// TIA Portal V20 export
VAR_GLOBAL   // PLC tag table "ConvConstantD1"
END_VAR
VAR_GLOBAL CONSTANT   // user constants
   minD1 : Int := 4001;
   maxD1 : Int := 4002;
END_VAR
